FUNCTION SingleSignalToLED : INT
VAR_INPUT
	LEDSignal	:	USINT;
END_VAR
VAR
END_VAR

// convert standard 0-255 LED signals to INT datatype
SingleSignalToLED := LEDSignal/256 * 32767;

END_FUNCTION

(* stored: Version 1.1.0.1, ProductVersion 3.1.4024.12
   POU SingleSignalToLED: Id {3cf7ba2c-e8e2-4a18-9731-d83d473d63c3}, SpecialFunc None *)
